DATA_BLOCK "DB_TT_TF_Type"
TITLE =%version: 0.10 % CN: 20
//History:
//This version  %created_by: nlhdl %
//              %date_created: Thursday, August 23, 2018 1:36:42 PM %
//              %release: VI_GEN/RA_Dev %
//
//Modification History:                                   By:    Date:     Rev:
//----------------------------------------------------  -------  --------  -----
//ra#30200: [ECS-P] Type DB not correct                 nlHdL    23-08-18   0.10
//ra#30200: Keep hardware with softstarter              nlHdL    20-08-18   0.09
//ra#30200: Modify FB_HW_MTR_TRI for movitrax           nlHdL    08-08-18   0.08
//ra#24152: TT LMS Error as LMS Not healthy             nlHdL    15-08-17   0.07
//ra#22982: Softstarter error during start up           nlHdL    19-06-17   0.06
//ra#20304: Asi error Status 19 wrong GS level          nlHdL    03-03-17   0.05
//ra#16735: DI NON_RETAIN PLC Memory                    nlHdL    13-12-16   0.04
//ra#15834: Added ASI and circuit breaker errors        nlDY     16-08-16   0.03
//ra#14800: Added errors and warnings                   nlDY     05-07-16   0.02
//Initial Revision based on version 0.07 TRS            nlHdL    08-06-16   0.01
//
FAMILY : General
VERSION : 0.0
NON_RETAIN

  STRUCT
   Type_Component : BYTE ;	//Type of the component (1 = Section, 0 = Other)
   Record_Length : BYTE ;	//Number of the Detailed Status in the UDT
   Status : ARRAY  [1 .. 48 ] OF "UDT_Comp_Status";
  END_STRUCT ;
BEGIN
   Type_Component := B#16#1;
   Record_Length := B#16#48;
   Status[1].HMI_Text_Number := -1;
   Status[1].Overall_Status_Relation := B#16#0;
   Status[1].General_Status_Relation := B#16#0;
   Status[2].HMI_Text_Number := -1;
   Status[2].Overall_Status_Relation := B#16#0;
   Status[2].General_Status_Relation := B#16#0;
   Status[3].HMI_Text_Number := -1;
   Status[3].Overall_Status_Relation := B#16#0;
   Status[3].General_Status_Relation := B#16#0;
   Status[4].HMI_Text_Number := -1;
   Status[4].Overall_Status_Relation := B#16#0;
   Status[4].General_Status_Relation := B#16#0;
   Status[5].HMI_Text_Number := -1;
   Status[5].Overall_Status_Relation := B#16#0;
   Status[5].General_Status_Relation := B#16#0;
   Status[6].HMI_Text_Number := -1;
   Status[6].Overall_Status_Relation := B#16#0;
   Status[6].General_Status_Relation := B#16#0;
   Status[7].HMI_Text_Number := -1;
   Status[7].Overall_Status_Relation := B#16#0;
   Status[7].General_Status_Relation := B#16#0;
   Status[8].HMI_Text_Number := -1;
   Status[8].Overall_Status_Relation := B#16#0;
   Status[8].General_Status_Relation := B#16#0;
   Status[9].HMI_Text_Number := 47;
   Status[9].Overall_Status_Relation := B#16#2;
   Status[9].General_Status_Relation := B#16#2;
   Status[10].HMI_Text_Number := 168;
   Status[10].Overall_Status_Relation := B#16#4;
   Status[10].General_Status_Relation := B#16#3;
   Status[11].HMI_Text_Number := 162;
   Status[11].Overall_Status_Relation := B#16#4;
   Status[11].General_Status_Relation := B#16#3;
   Status[12].HMI_Text_Number := 163;
   Status[12].Overall_Status_Relation := B#16#4;
   Status[12].General_Status_Relation := B#16#3;
   Status[13].HMI_Text_Number := 164;
   Status[13].Overall_Status_Relation := B#16#5;
   Status[13].General_Status_Relation := B#16#4;
   Status[14].HMI_Text_Number := 21;
   Status[14].Overall_Status_Relation := B#16#4;
   Status[14].General_Status_Relation := B#16#3;
   Status[15].HMI_Text_Number := 40;
   Status[15].Overall_Status_Relation := B#16#4;
   Status[15].General_Status_Relation := B#16#3;
   Status[16].HMI_Text_Number := 178;
   Status[16].Overall_Status_Relation := B#16#4;
   Status[16].General_Status_Relation := B#16#3;
   Status[17].HMI_Text_Number := 179;
   Status[17].Overall_Status_Relation := B#16#4;
   Status[17].General_Status_Relation := B#16#3;
   Status[18].HMI_Text_Number := 180;
   Status[18].Overall_Status_Relation := B#16#4;
   Status[18].General_Status_Relation := B#16#3;
   Status[19].HMI_Text_Number := 62;
   Status[19].Overall_Status_Relation := B#16#4;
   Status[19].General_Status_Relation := B#16#3;
   Status[20].HMI_Text_Number := 63;
   Status[20].Overall_Status_Relation := B#16#4;
   Status[20].General_Status_Relation := B#16#3;
   Status[21].HMI_Text_Number := 182;
   Status[21].Overall_Status_Relation := B#16#4;
   Status[21].General_Status_Relation := B#16#3;
   Status[22].HMI_Text_Number := 183;
   Status[22].Overall_Status_Relation := B#16#4;
   Status[22].General_Status_Relation := B#16#3;
   Status[23].HMI_Text_Number := 184;
   Status[23].Overall_Status_Relation := B#16#4;
   Status[23].General_Status_Relation := B#16#3;
   Status[24].HMI_Text_Number := 185;
   Status[24].Overall_Status_Relation := B#16#4;
   Status[24].General_Status_Relation := B#16#3;
   Status[25].HMI_Text_Number := 44;
   Status[25].Overall_Status_Relation := B#16#2;
   Status[25].General_Status_Relation := B#16#2;
   Status[26].HMI_Text_Number := 49;
   Status[26].Overall_Status_Relation := B#16#4;
   Status[26].General_Status_Relation := B#16#3;
   Status[27].HMI_Text_Number := 45;
   Status[27].Overall_Status_Relation := B#16#4;
   Status[27].General_Status_Relation := B#16#3;
   Status[28].HMI_Text_Number := 309;
   Status[28].Overall_Status_Relation := B#16#4;
   Status[28].General_Status_Relation := B#16#3;
   Status[29].HMI_Text_Number := 305;
   Status[29].Overall_Status_Relation := B#16#5;
   Status[29].General_Status_Relation := B#16#4;
   Status[30].HMI_Text_Number := 306;
   Status[30].Overall_Status_Relation := B#16#5;
   Status[30].General_Status_Relation := B#16#4;
   Status[31].HMI_Text_Number := 307;
   Status[31].Overall_Status_Relation := B#16#5;
   Status[31].General_Status_Relation := B#16#4;
   Status[32].HMI_Text_Number := 308;
   Status[32].Overall_Status_Relation := B#16#5;
   Status[32].General_Status_Relation := B#16#4;
   Status[33].HMI_Text_Number := 305;
   Status[33].Overall_Status_Relation := B#16#4;
   Status[33].General_Status_Relation := B#16#3;
   Status[34].HMI_Text_Number := 306;
   Status[34].Overall_Status_Relation := B#16#4;
   Status[34].General_Status_Relation := B#16#3;
   Status[35].HMI_Text_Number := 307;
   Status[35].Overall_Status_Relation := B#16#4;
   Status[35].General_Status_Relation := B#16#3;
   Status[36].HMI_Text_Number := 308;
   Status[36].Overall_Status_Relation := B#16#4;
   Status[36].General_Status_Relation := B#16#3;
   Status[37].HMI_Text_Number := 186;
   Status[37].Overall_Status_Relation := B#16#4;
   Status[37].General_Status_Relation := B#16#3;
   Status[38].HMI_Text_Number := 187;
   Status[38].Overall_Status_Relation := B#16#4;
   Status[38].General_Status_Relation := B#16#3;
   Status[39].HMI_Text_Number := -1;
   Status[39].Overall_Status_Relation := B#16#0;
   Status[39].General_Status_Relation := B#16#0;
   Status[40].HMI_Text_Number := -1;
   Status[40].Overall_Status_Relation := B#16#0;
   Status[40].General_Status_Relation := B#16#0;
   Status[41].HMI_Text_Number := -1;
   Status[41].Overall_Status_Relation := B#16#0;
   Status[41].General_Status_Relation := B#16#0;
   Status[42].HMI_Text_Number := -1;
   Status[42].Overall_Status_Relation := B#16#0;
   Status[42].General_Status_Relation := B#16#0;
   Status[43].HMI_Text_Number := -1;
   Status[43].Overall_Status_Relation := B#16#0;
   Status[43].General_Status_Relation := B#16#0;
   Status[44].HMI_Text_Number := -1;
   Status[44].Overall_Status_Relation := B#16#0;
   Status[44].General_Status_Relation := B#16#0;
   Status[45].HMI_Text_Number := -1;
   Status[45].Overall_Status_Relation := B#16#0;
   Status[45].General_Status_Relation := B#16#0;
   Status[46].HMI_Text_Number := -1;
   Status[46].Overall_Status_Relation := B#16#0;
   Status[46].General_Status_Relation := B#16#0;
   Status[47].HMI_Text_Number := -1;
   Status[47].Overall_Status_Relation := B#16#0;
   Status[47].General_Status_Relation := B#16#0;
   Status[48].HMI_Text_Number := -1;
   Status[48].Overall_Status_Relation := B#16#0;
   Status[48].General_Status_Relation := B#16#0;
END_DATA_BLOCK

